// TIA Portal V19 export
FUNCTION "MeasWheelCheckMechGearRatio" : Int   // FC19, LAD
TITLE = Use velocity of the measuring wheel for checking mechicak gear ratio of the motor
// Da usare per controllare i rapporti di riduzione impostati (esempio delle profilatrici)
// stored: Access Published, SetENOAutomatically false
   VAR_INPUT
      TO_Ax : TO_PositioningAxis;
      VelMin : LReal;
      ErrPercentageMax : LReal;
   END_VAR
   VAR_OUTPUT
      Err : LReal;
   END_VAR
   VAR_TEMP
      MeasWheelIsActive : Bool;
      ReductionRatio : LReal;
      MotorVelocity : LReal;
      MotorVelocityABS : LReal;
      ErrorPercentage : LReal;
      GearRatio : Bool;
      Check : Bool;
   END_VAR
   VAR CONSTANT
      RET_NULL : Int := 0;
      RET_VEL_OK : Int := 1;
      RET_VEL_BELOW_MIN : Int := 10;
      RET_ERR_ENC_NOT_VALID : Int := 101;
      RET_ERR_GEAR_RATIO : Int := 102;
      RET_VEL_DELTA_EXCEED : Int := 103;
   END_VAR
   VAR_TEMP   // added for the SCL form of the ladder/FBD networks
      _w1 : Bool;
   END_VAR
BEGIN

REGION Network 1: Out error percentage
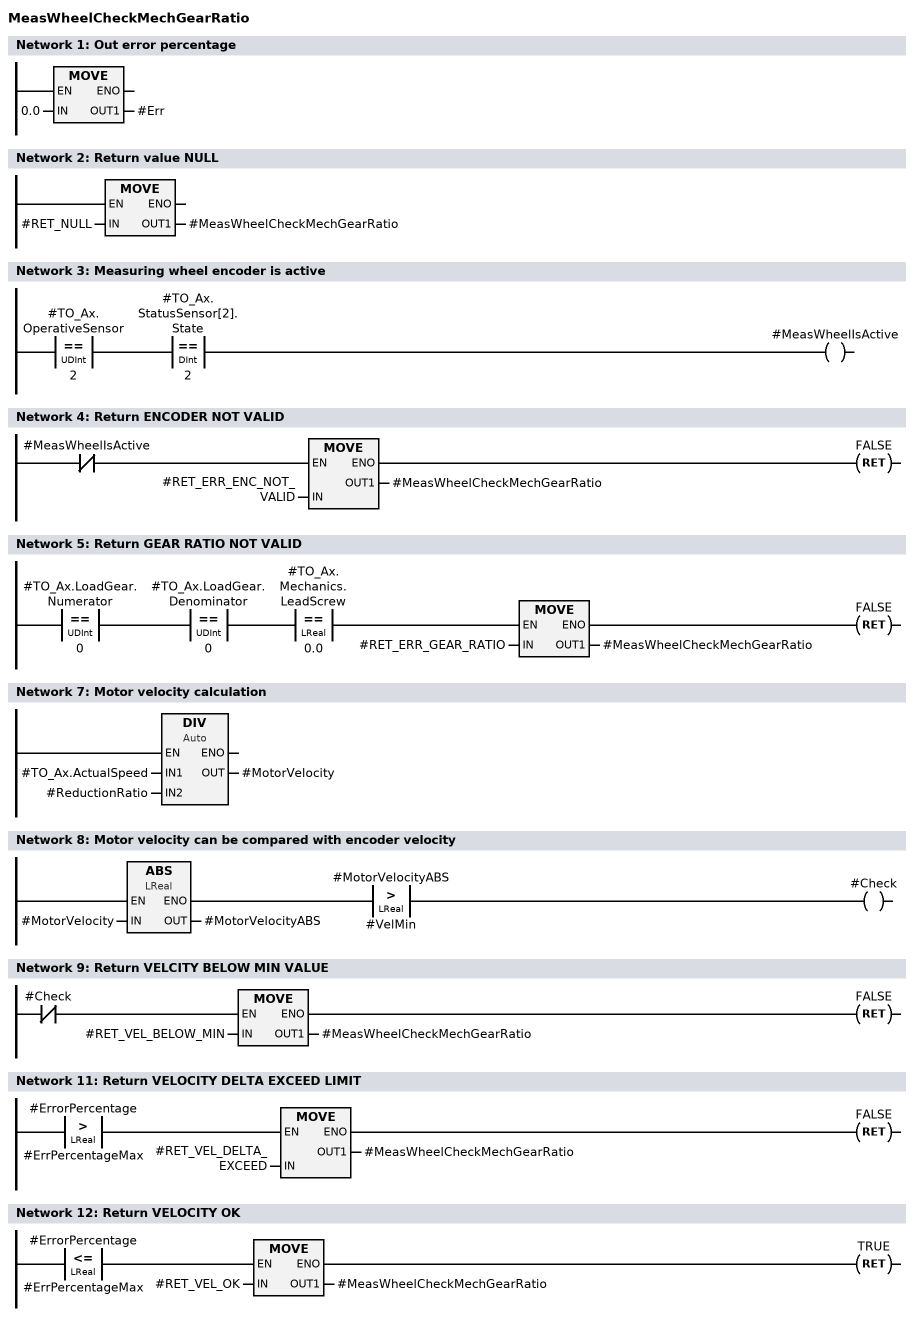
   RUNG wire#powerrail
      { S7_GenerateENO := "TRUE" } Move(in := 0.0, out1 => #Err)
   END_RUNG
   // the same network as SCL:
   #Err := 0.0;
END_REGION

REGION Network 2: Return value NULL
   RUNG wire#powerrail
      { S7_GenerateENO := "TRUE" } Move(in := #RET_NULL, out1 => #MeasWheelCheckMechGearRatio)
   END_RUNG
   // the same network as SCL:
   #MeasWheelCheckMechGearRatio := #RET_NULL;
END_REGION

REGION Network 3: Measuring wheel encoder is active
   RUNG wire#powerrail
      { S7_Templates := "SrcType := UDInt" } EQ_Contact(in1 := #TO_Ax.OperativeSensor, in2 := 2)
      { S7_Templates := "SrcType := DInt" } EQ_Contact(in1 := #TO_Ax.StatusSensor[2].State, in2 := 2)
      Coil( #MeasWheelIsActive )
   END_RUNG
   // the same network as SCL:
   #MeasWheelIsActive := (#TO_Ax.OperativeSensor = 2) AND (#TO_Ax.StatusSensor[2].State = 2);
END_REGION

REGION Network 4: Return ENCODER NOT VALID
   RUNG wire#powerrail
      I_Contact( #MeasWheelIsActive )
      Move(in := #RET_ERR_ENC_NOT_VALID, out1 => #MeasWheelCheckMechGearRatio)
      ReturnCoil( FALSE )
   END_RUNG
   // the same network as SCL:
   IF NOT #MeasWheelIsActive THEN
       #MeasWheelCheckMechGearRatio := #RET_ERR_ENC_NOT_VALID;
       ENO := FALSE;
       RETURN;
   END_IF;
END_REGION

REGION Network 5: Return GEAR RATIO NOT VALID
   // ENO of a box is taken as its EN; it also drops when the box reports an error
   #_w1 := (#TO_Ax.LoadGear.Numerator = 0) AND (#TO_Ax.LoadGear.Denominator = 0) AND (#TO_Ax.Mechanics.LeadScrew = 0.0);
   IF #_w1 THEN
       #MeasWheelCheckMechGearRatio := #RET_ERR_GEAR_RATIO;
       ENO := FALSE;
       RETURN;
   END_IF;
END_REGION

REGION Network 6 (SCL): Reuction ratio calculation

   #ReductionRatio := UDINT_TO_LREAL(#TO_Ax.LoadGear.Numerator / #TO_Ax.LoadGear.Denominator);

   #ReductionRatio := #TO_Ax.Mechanics.LeadScrew / #ReductionRatio;
END_REGION

REGION Network 7: Motor velocity calculation
   RUNG wire#powerrail
      Div(in1 := #TO_Ax.ActualSpeed, in2 := #ReductionRatio, out => #MotorVelocity)
   END_RUNG
   // the same network as SCL:
   #MotorVelocity := #TO_Ax.ActualSpeed / #ReductionRatio;
END_REGION

REGION Network 8: Motor velocity can be compared with encoder velocity
   RUNG wire#powerrail
      { S7_Templates := "SrcType := LReal"; S7_GenerateENO := "TRUE" } Abs(in := #MotorVelocity, out => #MotorVelocityABS)
      { S7_Templates := "SrcType := LReal" } GT_Contact(in1 := #MotorVelocityABS, in2 := #VelMin)
      Coil( #Check )
   END_RUNG
   // the same network as SCL:
   // ENO of a box is taken as its EN; it also drops when the box reports an error
   #MotorVelocityABS := ABS(#MotorVelocity);
   #Check := #MotorVelocityABS > #VelMin;
END_REGION

REGION Network 9: Return VELCITY BELOW MIN VALUE
   // ENO of a box is taken as its EN; it also drops when the box reports an error
   IF NOT #Check THEN
       #MeasWheelCheckMechGearRatio := #RET_VEL_BELOW_MIN;
       ENO := FALSE;
       RETURN;
   END_IF;
END_REGION

REGION Network 10 (SCL): Error percentage between motor and encoder

   #ErrorPercentage := ABS(100.0 * (#TO_Ax.StatusExtrapolation.ExtrapolatedVelocity - #MotorVelocity) / #MotorVelocity);


   #Err := #ErrorPercentage;
END_REGION

REGION Network 11: Return VELOCITY DELTA EXCEED LIMIT
   RUNG wire#powerrail
      { S7_Templates := "SrcType := LReal" } GT_Contact(in1 := #ErrorPercentage, in2 := #ErrPercentageMax)
      { S7_GenerateENO := "TRUE" } Move(in := #RET_VEL_DELTA_EXCEED, out1 => #MeasWheelCheckMechGearRatio)
      ReturnCoil( FALSE )
   END_RUNG
   // the same network as SCL:
   // ENO of a box is taken as its EN; it also drops when the box reports an error
   #_w1 := #ErrorPercentage > #ErrPercentageMax;
   IF #_w1 THEN
       #MeasWheelCheckMechGearRatio := #RET_VEL_DELTA_EXCEED;
       ENO := FALSE;
       RETURN;
   END_IF;
END_REGION

REGION Network 12: Return VELOCITY OK
   RUNG wire#powerrail
      { S7_Templates := "SrcType := LReal" } LE_Contact(in1 := #ErrorPercentage, in2 := #ErrPercentageMax)
      { S7_GenerateENO := "TRUE" } Move(in := #RET_VEL_OK, out1 => #MeasWheelCheckMechGearRatio)
      ReturnCoil( TRUE )
   END_RUNG
   // the same network as SCL:
   // ENO of a box is taken as its EN; it also drops when the box reports an error
   #_w1 := #ErrorPercentage <= #ErrPercentageMax;
   IF #_w1 THEN
       #MeasWheelCheckMechGearRatio := #RET_VEL_OK;
       ENO := TRUE;
       RETURN;
   END_IF;
END_REGION
END_FUNCTION
